{attribute addProperty BoxType "EJ7037-0000-0020"}
{attribute addProperty Id "StatusAT %I*Status_4F9ADA1B162"}
{attribute addProperty CRC "3414604698"}
{attribute addProperty SizeInBites "16"}
{attribute addProperty SizeInBytes "2"}
TYPE STM_Status_CB86BB9A :
STRUCT
	{attribute addProperty Name "Status"}
	Status AT %I* : Status_4F9ADA1B;
END_STRUCT
END_TYPE

(* stored: Version 1.2.0.0, ProductVersion 3.1.4024.9
   DUT STM_Status_CB86BB9A: Id {d8544cd1-a8e3-4a7d-aefe-3293e59671f4} *)
